// TwinCAT 3 PLC project Sample_PLC
// ProgramVersion: 3.1.4024.0
// libraries:
//   Tc2_MC2, * (Beckhoff Automation GmbH)
//   Tc2_Standard, * (Beckhoff Automation GmbH)
//   Tc2_System, * (Beckhoff Automation GmbH)
//   Tc2_Utilities, * (Beckhoff Automation GmbH)
//   Tc3_Module, * (Beckhoff Automation GmbH)
//   Tc3_TcForms, * (Kloetzer Automation)
// project tree:
//   GVLs/ GVL.TcGVL
//   / PlcTask.TcTTO
//   POUs/ FB_Gripper.TcPOU, MAIN.TcPOU, PRG_Automatic.TcPOU, PRG_NC_PTP.TcPOU
// real-time tasks:
//   TASK PlcTask: cycle T#10ms, priority 20, ADS port 350
// motion (NC):
//   TASK NC-Task 1 SAF: cycle T#2ms, priority 4, ADS port 501
//   TASK NC-Task 1 SVB: cycle T#10ms, priority 8, ADS port 511
//   AXIS X-Achse (id 1)
//     Dynamic: AccelerationMaximum=3000, DecelerationMaximum=3000, Acceleration=3000, Deceleration=3000, Jerk=30000
//     Velo: FastManual=300, Maximum=500
//     OtherSettings: AllowMotionCmdToSlave=true
//     encoder EncType=1
//     drive DrvType=5
//       Analog: VeloReferenz=500, TorqueSetpointScale=10, ScaleFactorActTorque=0.1
//       TimeComp: TaskDelayCycles=1
//     controller CtrType=1
//       CtrPara: PriorControlFactor=1
//         Observer: BandWidth=20
//   AXIS Y-Achse (id 2)
//     Dynamic: AccelerationMaximum=3000, DecelerationMaximum=3000, Acceleration=3000, Deceleration=3000, Jerk=30000
//     Velo: FastManual=300, Maximum=500
//     OtherSettings: AllowMotionCmdToSlave=true
//     encoder EncType=1
//     drive DrvType=5
//       Analog: VeloReferenz=500, TorqueSetpointScale=10, ScaleFactorActTorque=0.1
//       TimeComp: TaskDelayCycles=1
//     controller CtrType=1
//       CtrPara: PriorControlFactor=1
//         Observer: BandWidth=20
//   AXIS Z-Achse (id 3)
//     Dynamic: AccelerationMaximum=3000, DecelerationMaximum=3000, Acceleration=3000, Deceleration=3000, Jerk=30000
//     Velo: FastManual=300, Maximum=500
//     OtherSettings: AllowMotionCmdToSlave=true
//     encoder EncType=1
//     drive DrvType=5
//       Analog: VeloReferenz=500, TorqueSetpointScale=10, ScaleFactorActTorque=0.1
//       TimeComp: TaskDelayCycles=1
//     controller CtrType=1
//       CtrPara: PriorControlFactor=1
//         Observer: BandWidth=20
// variable links:
//   Sample PLC/Sample PLC Instance <-> NC-Task 1 SAF/Axes/X-Achse
//     PlcTask Inputs/PRG_NC_PTP.aAxisRef[1].NcToPlc <-> Outputs/ToPlc
//     PlcTask Outputs/PRG_NC_PTP.aAxisRef[1].PlcToNc <-> Inputs/FromPlc
//   Sample PLC/Sample PLC Instance <-> NC-Task 1 SAF/Axes/Y-Achse
//     PlcTask Inputs/PRG_NC_PTP.aAxisRef[2].NcToPlc <-> Outputs/ToPlc
//     PlcTask Outputs/PRG_NC_PTP.aAxisRef[2].PlcToNc <-> Inputs/FromPlc
//   Sample PLC/Sample PLC Instance <-> NC-Task 1 SAF/Axes/Z-Achse
//     PlcTask Inputs/PRG_NC_PTP.aAxisRef[3].NcToPlc <-> Outputs/ToPlc
//     PlcTask Outputs/PRG_NC_PTP.aAxisRef[3].PlcToNc <-> Inputs/FromPlc

CONFIGURATION Sample_PLC
    RESOURCE PLC ON TwinCAT3
        TASK PlcTask(INTERVAL := T#10ms, PRIORITY := 20);
        PROGRAM MAIN WITH PlcTask : MAIN;
    END_RESOURCE
END_CONFIGURATION

// ---- GVLs/GVL.TcGVL
{attribute 'qualified_only'}
VAR_GLOBAL
	
	bEnable				: BOOL;
	bReset				: BOOL;
	fOverride			: LREAL := 100;
	bFeedhold			: BOOL;
	bError				: BOOL;
	
	stEnable			: Tc3_TcForms.ST_SetResetCtrl;
	stStatus			: Tc3_TcForms.ST_SetResetState;
	
	aAxisStatus			: ARRAY[1..3] OF Tc3_TcForms.ST_LevelState;
	aAxisPowerEnable	: ARRAY[1..3] OF BOOL;
	aAxisPowerState		: ARRAY[1..3] OF Tc3_TcForms.ST_LevelState;
	aMoveAbsCtrl		: ARRAY[1..3] OF Tc3_TcForms.ST_EdgeTrigCtrl;
	aMoveAbsState		: ARRAY[1..3] OF Tc3_TcForms.ST_EdgeTrigState;
	aJogForward			: ARRAY[1..3] OF BOOL;
	aJogBackwards		: ARRAY[1..3] OF BOOL;
	bRapid				: BOOL;
	fInc				: LREAL := 1.0;
	bIncPlus			: BOOL;
	bIncMinus			: BOOL;
	
	stMoveAllCtrl		: Tc3_TcForms.ST_EdgeTrigCtrl;
	stMoveAllState		: Tc3_TcForms.ST_EdgeTrigState;
	
	stProgramCtrl		: Tc3_TcForms.ST_EdgeTrigCtrl;
	stProgramState		: Tc3_TcForms.ST_EdgeTrigState;
	nProgramState		: INT;
	nProgramStep		: INT;
	nProgramNo			: INT;
	
	aTargetPos			: ARRAY[1..3] OF LREAL;
	aActPos				: ARRAY[1..3] OF LREAL;
	
	bAirSupply			: BOOL;
	stGripperCtrl		: Tc3_TcForms.ST_SetResetCtrl;
	stGripperState		: Tc3_TcForms.ST_SetResetState;
	nGripperState		: INT;
	
	// Config
	fVelocity			: LREAL := 500.0;
	fPidKP				: LREAL := 10;
	fPidTn				: LREAL := 20.0;
	fPidTv				: LREAL := 0.0;


	bTest			: BOOL;
	nTestInt		: INT;
	nTestDint		: DINT;
	fTestLreal		: LREAL;
	sTest			: STRING(15);
	stTestCtrl		: Tc3_TcForms.ST_SetResetCtrl;
	stTestState		: Tc3_TcForms.ST_SetResetState;
	
	
	
END_VAR

// ---- POUs/MAIN.TcPOU
PROGRAM MAIN
VAR
	fbTcFormsLicense	: Tc3_TcForms.FB_License;
	
	i					: INT;
	rsEnable			: RS;
	tonEnable			: TON;
	tofEnable			: TOF;

	fbGripper			: FB_Gripper;
	
	nCnt 			: INT;
	nCalc 			: INT;
	
	rsTest			: RS;
	tonTest			: TON;
	tofTest			: TOF;
END_VAR

// TcForms License
fbTcFormsLicense(bExecute:=TRUE);

// Global Enable
rsEnable(SET:=GVL.stEnable.bSet, RESET1:=GVL.stEnable.bReset, Q1=>GVL.bEnable);
tonEnable(IN:=GVL.bEnable, PT:=T#1S);
tofEnable(IN:=GVL.bEnable, PT:=T#1S);
GVL.stStatus.bDone := GVL.stEnable.bSet OR GVL.stEnable.bReset;
GVL.stStatus.bBusy := GVL.bEnable;
GVL.stStatus.bOn := TRUE;
GVL.stStatus.bOff := TRUE;
FOR i:=1 TO 3 DO
	GVL.aAxisPowerEnable[i] S= GVL.stEnable.bSet;
	GVL.aAxisPowerEnable[i] R= GVL.stEnable.bReset;
	GVL.stStatus.bOn := GVL.stStatus.bOn AND GVL.aAxisPowerState[i].bStatus;
	GVL.stStatus.bOff := GVL.stStatus.bOff AND NOT GVL.aAxisPowerState[i].bStatus;
END_FOR
GVL.bAirSupply S= GVL.stEnable.bSet;
GVL.bAirSupply R= GVL.stEnable.bReset;
GVL.stStatus.bOn := GVL.stStatus.bOn AND GVL.bAirSupply;
GVL.stStatus.bOff := GVL.stStatus.bOff AND NOT GVL.bAirSupply;
GVL.stStatus.bError := (tonEnable.Q AND NOT GVL.stStatus.bOn) OR (NOT tofEnable.Q AND NOT GVL.stStatus.bOff);
// -----------------------------------------------------------------

// Automatic
PRG_Automatic();
// -----------------------------------------------------------------

// NC PTP
PRG_NC_PTP();
// -----------------------------------------------------------------

// Gripper
fbGripper(bAirSupply:=GVL.bAirSupply, stCtrl:=GVL.stGripperCtrl, stState=>GVL.stGripperState);
IF GVL.stGripperState.bOn THEN
	GVL.nGripperState := 2;
ELSIF GVL.stGripperState.bOff THEN
	GVL.nGripperState := 1;
ELSE
	GVL.nGripperState := 0;
END_IF
// -----------------------------------------------------------------

// Global Error / Error Reset
GVL.bError := GVL.stStatus.bError OR
			  GVL.aAxisStatus[1].bError OR GVL.aAxisStatus[2].bError OR GVL.aAxisStatus[3].bError OR			  
			  GVL.aAxisPowerState[1].bError OR GVL.aAxisPowerState[2].bError OR GVL.aAxisPowerState[3].bError OR
			  GVL.aMoveAbsState[1].bError OR GVL.aMoveAbsState[2].bError OR GVL.aMoveAbsState[3].bError OR
			  GVL.stProgramState.bError OR
			  GVL.stGripperState.bError;
			  
GVL.bReset := FALSE;





nCnt := nCnt + 1;
GVL.bTest := GVL.bTest;
GVL.nTestDint := GVL.nTestDint;
GVL.fTestLreal := GVL.fTestLreal;	
	
rsTest(SET:=GVL.stTestCtrl.bSet,RESET1:=GVL.stTestCtrl.bReset,Q1=>GVL.stTestState.bBusy);
GVL.stTestState.bDone := GVL.stTestCtrl.bSet OR GVL.stTestCtrl.bReset;
tonTest(IN:=rsTest.Q1,PT:=T#2S);
tofTest(IN:=rsTest.Q1,PT:=T#2S);
GVL.stTestState.bOn := tonTest.Q;
GVL.stTestState.bOff := NOT tofTest.Q;

END_PROGRAM

// ---- POUs/FB_Gripper.TcPOU
FUNCTION_BLOCK FB_Gripper
VAR_INPUT
	bAirSupply	: BOOL;
	stCtrl		: Tc3_TcForms.ST_SetResetCtrl;
END_VAR
VAR_OUTPUT
	stState		: Tc3_TcForms.ST_SetResetState;
END_VAR
VAR
	rsGripper			: RS;
	tonGripper			: TON;
	tofGripper			: TOF;
	tonError			: TON;
	rtErrorAck			: R_TRIG;
END_VAR

rsGripper(SET:=stCtrl.bSet,RESET1:=stCtrl.bReset,Q1=>stState.bBusy);
tonGripper(IN:=rsGripper.Q1 AND bAirSupply,PT:=T#1S);
tofGripper(IN:=rsGripper.Q1 AND bAirSupply,PT:=T#1S);
stState.bOn := tonGripper.Q;
stState.bOff := NOT tofGripper.Q;
tonError(IN:=(stState.bBusy AND stState.bOff) OR (NOT stState.bBusy AND stState.bOn),PT:=T#2S,Q=>stState.bError);
stState.bDone := stCtrl.bSet OR stCtrl.bReset;
rtErrorAck(CLK:=stState.bDone);
IF rtErrorAck.Q THEN
	tonError(IN:=FALSE);
END_IF

END_FUNCTION_BLOCK

// ---- POUs/PRG_Automatic.TcPOU
PROGRAM PRG_Automatic
VAR
	nState				: INT;
	rtExecute			: R_TRIG;
	rtAbort				: R_TRIG;
	nNumberOfParts		: INT;
	nCounter			: INT;
	i					: INT;
	bNotBusy			: BOOL;
	bError				: bool;
END_VAR
VAR CONSTANT
	Z_UP				: LREAL := 200.0;
	Z_DOWN				: LREAL := 0.0;
	X1					: LREAL := 500.0;
	Y1					: LREAL := 500.0;
	X2					: LREAL := -300.0;
	Y2					: LREAL := -300.0;
	NUMBER_OF_PARTS		: ARRAY[0..2] OF INT := [3, 5, 10];
END_VAR

rtExecute(CLK:=GVL.stProgramCtrl.bExecute);
rtAbort(CLK:=GVL.stProgramCtrl.bAbort);
GVL.stProgramCtrl.bExecute R= GVL.bReset;
GVL.stProgramCtrl.bAbort R= GVL.bReset;
IF nState>0 AND (rtAbort.Q OR GVL.bReset OR GVL.bError) THEN
	bError := GVL.bError;
	nState := -1;
END_IF

CASE nState OF
	-1:		// Abort
		bNotBusy := TRUE;	
		FOR i:=1 TO 3 DO
			GVL.aMoveAbsCtrl[i].bAbort := TRUE;
			bNotBusy := bNotBusy AND NOT GVL.aMoveAbsState[i].bBusy;
		END_FOR
		IF bNotBusy THEN
			FOR i:=1 TO 3 DO
				GVL.aMoveAbsCtrl[i].bExecute := FALSE;
				GVL.aMoveAbsCtrl[i].bAbort := FALSE;
			END_FOR
			GVL.stProgramState.bBusy := FALSE;
			GVL.stProgramState.bAborted := NOT bError;
			GVL.stProgramState.bError := bError;
			nState := 0;
		END_IF
		
	0:		// Idle
		IF rtExecute.Q THEN
			nNumberOfParts := NUMBER_OF_PARTS[GVL.nProgramNo];
			nCounter := 0;
			GVL.stProgramState.bBusy := TRUE;
			nState := nState + 1;
		ELSIF NOT GVL.stProgramCtrl.bExecute THEN
			bError := FALSE;
			GVL.stProgramState.nErrorId := 0;
			GVL.stProgramState.bError := FALSE;
			GVL.stProgramState.bBusy := FALSE;
			GVL.stProgramState.bAborted := FALSE;
			GVL.stProgramState.bDone := FALSE;
		END_IF
		
	1:		// Open Gripper
		GVL.stGripperCtrl.bReset := TRUE;
		IF GVL.stGripperState.bDone AND GVL.stGripperState.bOff THEN
			GVL.stGripperCtrl.bReset := FALSE;
			nState := nState + 1;
		ELSIF GVL.stGripperState.bError THEN
			bError := TRUE;
			GVL.stProgramState.nErrorId := INT_TO_UDINT(nState);
			nState := -1;
		END_IF
		
	2:		// Move Z up
		GVL.aTargetPos[3] := Z_UP;
		GVL.aMoveAbsCtrl[3].bExecute := TRUE;
		IF GVL.aMoveAbsState[3].bDone THEN
			GVL.aMoveAbsCtrl[3].bExecute := FALSE;
			nState := nState + 1;
		ELSIF GVL.aMoveAbsState[3].bError OR GVL.aMoveAbsState[3].bAborted THEN
			bError := TRUE;
			GVL.stProgramState.nErrorId := INT_TO_UDINT(nState);
			nState := -1;
		END_IF
		
	3:		// Move to Pos 1
		GVL.aTargetPos[1] := X1;
		GVL.aTargetPos[2] := Y1;
		GVL.aMoveAbsCtrl[1].bExecute := TRUE;
		GVL.aMoveAbsCtrl[2].bExecute := TRUE;
		IF GVL.aMoveAbsState[1].bDone AND GVL.aMoveAbsState[2].bDone THEN
			GVL.aMoveAbsCtrl[1].bExecute := FALSE;
			GVL.aMoveAbsCtrl[2].bExecute := FALSE;
			nState := nState + 1;
		ELSIF GVL.aMoveAbsState[1].bError OR GVL.aMoveAbsState[1].bAborted OR 
			  GVL.aMoveAbsState[2].bError OR GVL.aMoveAbsState[2].bAborted THEN
			bError := TRUE;
			GVL.stProgramState.nErrorId := INT_TO_UDINT(nState);
			nState := -1;
		END_IF
		
	4:		// Move Z down
		GVL.aTargetPos[3] := Z_DOWN;
		GVL.aMoveAbsCtrl[3].bExecute := TRUE;
		IF GVL.aMoveAbsState[3].bDone THEN
			GVL.aMoveAbsCtrl[3].bExecute := FALSE;
			nState := nState + 1;
		ELSIF GVL.aMoveAbsState[3].bError OR GVL.aMoveAbsState[3].bAborted THEN
			bError := TRUE;
			GVL.stProgramState.nErrorId := INT_TO_UDINT(nState);
			nState := -1;
		END_IF
		
	5:		// Close Gripper
		GVL.stGripperCtrl.bSet := TRUE;
		IF GVL.stGripperState.bDone AND GVL.stGripperState.bOn THEN
			GVL.stGripperCtrl.bSet := FALSE;
			nState := nState + 1;
		ELSIF GVL.stGripperState.bError THEN
			bError := TRUE;
			GVL.stProgramState.nErrorId := INT_TO_UDINT(nState);
			nState := -1;
		END_IF
		
	6:		// Move Z up
		GVL.aTargetPos[3] := Z_UP;
		GVL.aMoveAbsCtrl[3].bExecute := TRUE;
		IF GVL.aMoveAbsState[3].bDone THEN
			GVL.aMoveAbsCtrl[3].bExecute := FALSE;
			nState := nState + 1;
		ELSIF GVL.aMoveAbsState[3].bError OR GVL.aMoveAbsState[3].bAborted THEN
			bError := TRUE;
			GVL.stProgramState.nErrorId := INT_TO_UDINT(nState);
			nState := -1;
		END_IF
		
	7:		// Move to Pos 2
		GVL.aTargetPos[1] := X2;
		GVL.aTargetPos[2] := Y2;
		GVL.aMoveAbsCtrl[1].bExecute := TRUE;
		GVL.aMoveAbsCtrl[2].bExecute := TRUE;
		IF GVL.aMoveAbsState[1].bDone AND GVL.aMoveAbsState[2].bDone THEN
			GVL.aMoveAbsCtrl[1].bExecute := FALSE;
			GVL.aMoveAbsCtrl[2].bExecute := FALSE;
			nState := nState + 1;
		ELSIF GVL.aMoveAbsState[1].bError OR GVL.aMoveAbsState[1].bAborted OR 
			  GVL.aMoveAbsState[2].bError OR GVL.aMoveAbsState[2].bAborted THEN			
			bError := TRUE;
			GVL.stProgramState.nErrorId := INT_TO_UDINT(nState);
			nState := -1;
		END_IF
		
	8:		// Move Z down
		GVL.aTargetPos[3] := Z_DOWN;
		GVL.aMoveAbsCtrl[3].bExecute := TRUE;
		IF GVL.aMoveAbsState[3].bDone THEN
			GVL.aMoveAbsCtrl[3].bExecute := FALSE;
			nState := nState + 1;
		ELSIF GVL.aMoveAbsState[3].bError OR GVL.aMoveAbsState[3].bAborted THEN
			bError := TRUE;
			GVL.stProgramState.nErrorId := INT_TO_UDINT(nState);
			nState := -1;
		END_IF
		
	9:		// Open Gripper
		GVL.stGripperCtrl.bReset := TRUE;
		IF GVL.stGripperState.bDone AND GVL.stGripperState.bOff THEN
			GVL.stGripperCtrl.bReset := FALSE;
			nState := nState + 1;
			nCounter := nCounter + 1;
		ELSIF GVL.stGripperState.bError THEN
			bError := TRUE;
			GVL.stProgramState.nErrorId := INT_TO_UDINT(nState);
			nState := -1;
		END_IF
		
	10:
		IF nCounter = nNumberOfParts THEN
			GVL.stProgramState.bBusy := FALSE;
			GVL.stProgramState.bDone := TRUE;
			nState := 0;
		ELSE
			nState := 1;
		END_IF
		
	
END_CASE

GVL.nProgramStep := nState + 1;

IF GVL.stProgramState.bError THEN
	GVL.nProgramState := 4;
ELSIF GVL.stProgramState.bAborted THEN
	GVL.nProgramState := 3;
ELSIF GVL.stProgramState.bDone THEN
	GVL.nProgramState := 2;
ELSIF GVL.stProgramState.bBusy THEN
	GVL.nProgramState := 1;
ELSE
	GVL.nProgramState := 0;
END_IF

END_PROGRAM

// ---- POUs/PRG_NC_PTP.TcPOU
PROGRAM PRG_NC_PTP
VAR
	i				: INT;
	aAxisRef		: ARRAY[1..3] OF AXIS_REF;
	mcPower			: ARRAY[1..3] OF MC_Power;
	mcReset			: ARRAY[1..3] OF MC_Reset;
	mcMoveAbsolute	: ARRAY[1..3] OF MC_MoveAbsolute;
	mcHalt			: ARRAY[1..3] OF MC_Halt;
	mcJog			: ARRAY[1..3] OF MC_Jog;
	tonJogForward	: ARRAY[1..3] OF TON;
	tonJogBackwards	: ARRAY[1..3] OF TON;
	ftJogForward	: ARRAY[1..3] OF F_TRIG;
	ftJogBackwards	: ARRAY[1..3] OF F_TRIG;
	rtAbort			: ARRAY[1..3] OF R_TRIG;
	rtExecMoveAll	: R_TRIG;
END_VAR

rtExecMoveAll(CLK:=GVL.stMoveAllCtrl.bExecute);
GVL.stMoveAllCtrl.bExecute R= GVL.bReset;
GVL.stMoveAllCtrl.bAbort R= GVL.bReset;
IF rtExecMoveAll.Q THEN
	GVL.stMoveAllState.bBusy := TRUE;
	GVL.aMoveAbsCtrl[1].bExecute := TRUE;
	GVL.aMoveAbsCtrl[2].bExecute := TRUE;
	GVL.aMoveAbsCtrl[3].bExecute := TRUE;
ELSIF GVL.stMoveAllState.bBusy THEN
	GVL.stMoveAllState.bDone := GVL.aMoveAbsState[1].bDone AND GVL.aMoveAbsState[2].bDone AND GVL.aMoveAbsState[3].bDone;
	GVL.stMoveAllState.bError := GVL.aMoveAbsState[1].bError OR GVL.aMoveAbsState[2].bError OR GVL.aMoveAbsState[3].bError;
	GVL.stMoveAllState.bAborted := (NOT GVL.aMoveAbsState[1].bBusy AND NOT GVL.aMoveAbsState[2].bBusy AND NOT GVL.aMoveAbsState[3].bBusy AND GVL.stMoveAllCtrl.bAbort);
	GVL.stMoveAllState.bBusy R= (NOT GVL.aMoveAbsState[1].bBusy AND NOT GVL.aMoveAbsState[2].bBusy AND NOT GVL.aMoveAbsState[3].bBusy);
	GVL.aMoveAbsCtrl[1].bAbort S= GVL.stMoveAllCtrl.bAbort OR (GVL.stMoveAllState.bError AND GVL.aMoveAbsState[1].bBusy);
	GVL.aMoveAbsCtrl[2].bAbort S= GVL.stMoveAllCtrl.bAbort OR (GVL.stMoveAllState.bError AND GVL.aMoveAbsState[2].bBusy);
	GVL.aMoveAbsCtrl[3].bAbort S= GVL.stMoveAllCtrl.bAbort OR (GVL.stMoveAllState.bError AND GVL.aMoveAbsState[3].bBusy);
ELSIF NOT GVL.stMoveAllCtrl.bExecute AND (GVL.stMoveAllState.bDone OR GVL.stMoveAllState.bError OR GVL.stMoveAllState.bAborted) THEN
	GVL.stMoveAllState.bDone := FALSE;
	GVL.stMoveAllState.bError := FALSE;
	GVL.stMoveAllState.bAborted := FALSE;
	GVL.aMoveAbsCtrl[1].bExecute := FALSE;
	GVL.aMoveAbsCtrl[2].bExecute := FALSE;
	GVL.aMoveAbsCtrl[3].bExecute := FALSE;
	GVL.aMoveAbsCtrl[1].bAbort := FALSE;
	GVL.aMoveAbsCtrl[2].bAbort := FALSE;
	GVL.aMoveAbsCtrl[3].bAbort := FALSE;
END_IF




FOR i:=1 TO 3 DO
	
	aAxisRef[i].ReadStatus();
	GVL.aAxisStatus[i].bError := aAxisRef[i].Status.Error;
	GVL.aAxisStatus[i].nErrorId := aAxisRef[i].Status.ErrorID;
	
	mcPower[i](
		Axis:= aAxisRef[i], 
		Enable:= GVL.aAxisPowerEnable[i], 
		Enable_Positive:= TRUE, 
		Enable_Negative:= TRUE, 
		Override:= GVL.fOverride*BOOL_TO_LREAL(NOT GVL.bFeedhold), 
		BufferMode:= , 
		Options:= , 
		Status=> GVL.aAxisPowerState[i].bStatus, 
		Busy=> GVL.aAxisPowerState[i].bBusy,  
		Active=> GVL.aAxisPowerState[i].bActive, 
		Error=> GVL.aAxisPowerState[i].bError,  
		ErrorID=> );
		
	mcReset[i](
		Axis:= aAxisRef[i], 
		Execute:= GVL.bReset AND aAxisRef[i].Status.Error,
		Done=> , 
		Busy=> , 
		Error=> ,  
		ErrorID=> );
		
	mcMoveAbsolute[i](
		Axis:= aAxisRef[i],
		Execute:= GVL.aMoveAbsCtrl[i].bExecute, 
		Position:= GVL.aTargetPos[i], 
		Velocity:= GVL.fVelocity, 
		Acceleration:= , 
		Deceleration:= , 
		Jerk:= , 
		BufferMode:= , 
		Options:= , 
		Done=> GVL.aMoveAbsState[i].bDone, 
		Busy=> GVL.aMoveAbsState[i].bBusy,  
		Active=> GVL.aMoveAbsState[i].bActive,  
		CommandAborted=> GVL.aMoveAbsState[i].bAborted, 
		Error=> GVL.aMoveAbsState[i].bError, 
		ErrorID=> GVL.aMoveAbsState[i].nErrorId);
	GVL.aMoveAbsCtrl[i].bExecute R= GVL.bReset;
		
	rtAbort[i](CLK:=GVL.aMoveAbsCtrl[i].bAbort);
	mcHalt[i](
		Axis:= aAxisRef[i],
		Execute:= rtAbort[i].Q OR GVL.bReset, 
		Deceleration:= , 
		Jerk:= , 
		BufferMode:= , 
		Options:= , 
		Done=> , 
		Busy=> , 
		Active=> , 
		CommandAborted=> , 
		Error=> , 
		ErrorID=> );
	GVL.aMoveAbsCtrl[i].bAbort R= GVL.bReset;
		
	IF NOT GVL.stProgramState.bBusy THEN
		
		GVL.aJogForward[i] := GVL.aJogForward[i] AND NOT GVL.bFeedhold;
		GVL.aJogBackwards[i] := GVL.aJogBackwards[i] AND NOT GVL.bFeedhold;
		tonJogForward[i](IN:=GVL.aJogForward[i],PT:=T#500MS);
		tonJogBackwards[i](IN:=GVL.aJogBackwards[i],PT:=T#500MS);
		ftJogForward[i](CLK:=NOT tonJogForward[i].Q AND GVL.aJogForward[i]);
		ftJogBackwards[i](CLK:=NOT tonJogBackwards[i].Q AND GVL.aJogBackwards[i]);
		IF tonJogForward[i].Q OR tonJogBackwards[i].Q THEN
			IF GVL.bRapid THEN
				mcJog[i].Mode := E_JogMode.MC_JOGMODE_STANDARD_FAST;
			ELSE
				mcJog[i].Mode := E_JogMode.MC_JOGMODE_STANDARD_SLOW;
			END_IF
			mcJog[i].JogForward := tonJogForward[i].Q;
			mcJog[i].JogBackwards := tonJogBackwards[i].Q;
			mcJog[i].Velocity := 500.0;
		ELSE
			mcJog[i].Mode := E_JogMode.MC_JOGMODE_INCHING;
			mcJog[i].Velocity := 100.0;
			mcJog[i].JogForward := ftJogForward[i].Q;
			mcJog[i].JogBackwards := ftJogBackwards[i].Q;
		END_IF
		
		mcJog[i](
			Axis:= aAxisRef[i],
	//		JogForward:= GVL.aJogForward[i],
	//		JogBackwards:= GVL.aJogBackwards[i], 
	//		Mode:= E_JogMode.MC_JOGMODE_STANDARD_FAST, 
			Position:= GVL.fInc, 
	//		Velocity:= 100.0, 
			Acceleration:= , 
			Deceleration:= , 
			Jerk:= , 
			Done=> , 
			Busy=> , 
			Active=> , 
			CommandAborted=> , 
			Error=> , 
			ErrorID=> );
	
	END_IF
		
	GVL.aActPos[i] := aAxisRef[i].NcToPlc.ActPos;
	
END_FOR

IF GVL.bIncPlus AND GVL.fInc<=10.0 THEN
	GVL.fInc := GVL.fInc * 10.0;	
ELSIF GVL.bIncMinus AND GVL.fInc>=0.01 THEN
	GVL.fInc := GVL.fInc / 10.0;
END_IF
GVL.bIncPlus := FALSE;
GVL.bIncMinus := FALSE;

END_PROGRAM
